FUNCTION_BLOCK FB_TelescopeReferencingState EXTENDS FB_TelescopeState
VAR_INPUT
END_VAR
VAR_OUTPUT
END_VAR
VAR
END_VAR

END_FUNCTION_BLOCK

(* stored: Version 1.1.0.1, ProductVersion 3.1.4024.15
   POU FB_TelescopeReferencingState: Id {3471d165-9b96-4b1b-90bd-c2a75cfe669b}, SpecialFunc None *)
